Universal Robots PolyScope program: sockets3enrayadefinitivo.urp

Program sockets3enrayadefinitivo (installation=default directory=/programs/Alumnes/Arnau/Raya createdIn=5.17.3 lastSavedIn=5.20.0 robotSerialNumber=20205300829)
Calibrated DH parameters: a=[0.000012, -0.242852, -0.179835, 0.000093, -0.000124, 0]; d=[0.151981, 5.088974, 36.181125, -41.139477, 0.085414, 0.092081]; alpha=[1.572112, -0.003585, 0.002783, 1.571586, -1.572466, 0]; deltaTheta=[0, -0.074993, 0.643315, -0.56833, 0.000002, 0]
InitVariablesNode
BeforeStart
  Script file /programs/Alumnes/Arnau/Raya/pepe.script_bak
    | # Función para calcular la posición en el tablero 3x3
    | def calcular_posicion(base_pos, cell_num, paso_x, paso_y):
    |     fila = floor((cell_num - 1) / 3)
    |     columna = (cell_num - 1) % 3
    | 
    |     nueva_x = base_pos[0] + (columna * paso_x)
    |     nueva_y = base_pos[1] - (fila * paso_y)
    |     nueva_z = base_pos[2]
    | 
    |     return p[nueva_x, nueva_y, nueva_z, base_pos[3], base_pos[4], base_pos[5]]
    | end
    | 
    | def calcular_posicion_arriba(base_pos, cell_num, paso_x, paso_y):
    |     fila = floor((cell_num - 1) / 3)
    |     columna = (cell_num - 1) % 3
    | 
    |     nueva_x = base_pos[0] + (columna * paso_x)
    |     nueva_y = base_pos[1] - (fila * paso_y)
    |     nueva_z = base_pos[2] + 0.1
    | 
    |     return p[nueva_x, nueva_y, nueva_z, base_pos[3], base_pos[4], base_pos[5]]
    | end
    | # Función para obtener el número de un string "num letra"
    | def obtener_numero(texto):
    |     espacio = str_find(texto, " ")
    |     if espacio < 0:
    |         return -1  # Manejo de error si no hay espacio
    |     end
    |     num_str = str_sub(texto, 0, espacio)
    |     return to_num(num_str)
    | end
    | 
    | # Función para obtener la ficha ("X" o "O") de un string "num letra"
    | def obtener_ficha(texto):
    |     espacio = str_find(texto, " ")
    |     if espacio < 0:
    |         return ""  # Manejo de error si no hay espacio
    |     end
    |     return str_sub(texto, espacio + 1, str_len(texto))
    | end
    | 
    | # Función para calcular la posición de una ficha en el tablero 2x5
    | def calcular_posicion_ficha(base_pos, cantidad_restante, paso_x, paso_y):
    |     # Calcular la columna y la fila
    |     columna = floor((10 - cantidad_restante) / 2)  # Cambia cada 2 fichas
    |     fila = (cantidad_restante+1) % 2  # Alterna entre 0 y 1
    | 
    |     # Calcular nueva posición
    |     nueva_x = base_pos[0] + (columna * paso_x)
    |     nueva_y = base_pos[1] - (fila * paso_y)
    |     nueva_z = base_pos[2]
    | 
    |     return p[nueva_x, nueva_y, nueva_z, base_pos[3], base_pos[4], base_pos[5]]
    | end
    | 
    | def calcular_posicion_ficha_arriba(base_pos, cantidad_restante, paso_x, paso_y):
    |     # Calcular la columna y la fila
    |     columna = floor((10 - cantidad_restante) / 2)  # Cambia cada 2 fichas
    |     fila = (cantidad_restante +1) % 2  # Alterna entre 0 y 1
    | 
    |     # Calcular nueva posición
    |     nueva_x = base_pos[0] + (columna * paso_x)
    |     nueva_y = base_pos[1] - (fila * paso_y)
    |     nueva_z = base_pos[2] +0.1
    | 
    |     return p[nueva_x, nueva_y, nueva_z, base_pos[3], base_pos[4], base_pos[5]]
    | end
  restantes := 10
  paso_tablero := 0.07
  paso_x_fichas := 0.052
  paso_y_fichas := 0.07
  posi_tablero := p[0.250183,-0.0555376,0.00556842,-2.307,2.12022,-0.0152373]
  posi_fichas := p[0.218027,0.168794,0.00429337,2.24033,-2.20236,1.95739e-05]
  socket := socket_open("172.30.3.77", 5858, "s1")
Robot Program (runOnlyOnce=false)
  Loop While (checkContinuously=false) expression=socket≟ False
    socket := socket_open("172/30.3.77", 5858, "s1")
  input := socket_read_string("s1",timeout=2)
  MoveJ speed 60 deg/s, acceleration 80 deg/s^2 (useActiveTCP=true) feature=Base
    Waypoint Waypoint_1: TCP in base x=228.93 y=40.681 z=141.238 mm, rx=2.9899 ry=-0.9644 rz=0 rad; joints [-204.591, -115.74, 109.647, -84.002, 270.321, 281.367] deg; TCP offset x=0 y=0 z=160 mm, rx=0 ry=0 rz=0 rad
  URCap 2FG Release (OnRobot, OnRobot A/S) dataModel(twofg.external-grip.target-width=0.07100000000000001, twofg.internal-grip.target-width=0.085)
  Loop While (checkContinuously=false) expression=input≟""
    input := socket_read_string("s1",timeout=2)
    Wait Sleep waitTime=1
  Script: movel(calcular_posicion_ficha_arriba(posi_fichas,restantes,paso_x_fichas,paso_y_fichas),1.2,0.25,0,0)
  Script: movel(calcular_posicion_ficha(posi_fichas,restantes,paso_x_fichas,paso_y_fichas),1.2,0.25,0,0)
  URCap 2FG Grip (OnRobot, OnRobot A/S) dataModel(twofg.target-speed=50, twofg.target-force=20, twofg.external-grip.target-width=0.033, twofg.internal-grip.target-width=0.047)
  Script: movel(calcular_posicion_ficha_arriba(posi_fichas,restantes,paso_x_fichas,paso_y_fichas),1.2,0.25,0,0)
  restantes := restantes-1
  Script: movel(calcular_posicion_arriba(posi_tablero,obtener_numero(input),paso_tablero,paso_tablero),1.2,0.25,0,0)
  Script: movel(calcular_posicion(posi_tablero,obtener_numero(input),paso_tablero,paso_tablero),1.2,0.25,0,0)
  URCap 2FG Release (OnRobot, OnRobot A/S) dataModel(twofg.external-grip.target-width=0.07, twofg.internal-grip.target-width=0.084, twofg.target-speed=51)
  Script: movel(calcular_posicion_arriba(posi_tablero,obtener_numero(input),paso_tablero,paso_tablero),1.2,0.25,0,0)
